// SIMATIC S7-200 SMART project (STEP 7-Micro/WIN SMART), CPU SR40

SYMBOL_TABLE 系统符号
Clock_1s         SM0.5    // 针对 1 s 的周期时间，时钟脉冲接通 0.5 s，断开 0.5 s.
END_SYMBOL_TABLE

ORGANIZATION_BLOCK MAIN:OB1
TITLE=程序注释
BEGIN
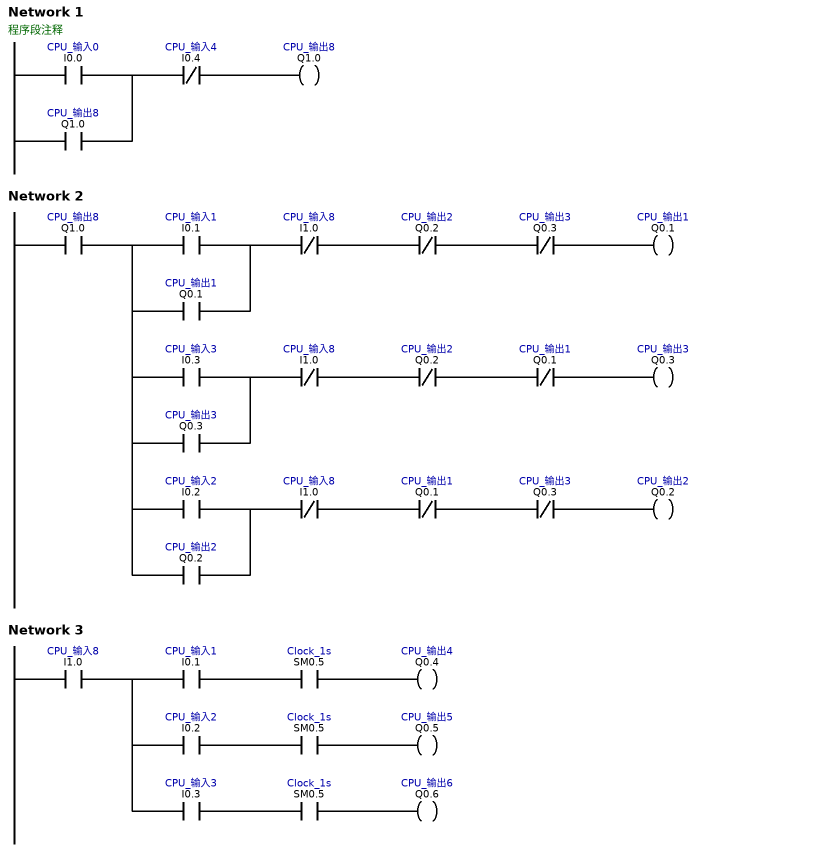
Network 1
// 程序段注释
LD     CPU_输入0:I0.0
O      CPU_输出8:Q1.0
AN     CPU_输入4:I0.4
=      CPU_输出8:Q1.0
Network 2
LD     CPU_输出8:Q1.0
LPS
LD     CPU_输入1:I0.1
O      CPU_输出1:Q0.1
ALD
AN     CPU_输入8:I1.0
AN     CPU_输出2:Q0.2
AN     CPU_输出3:Q0.3
=      CPU_输出1:Q0.1
LRD
LD     CPU_输入3:I0.3
O      CPU_输出3:Q0.3
ALD
AN     CPU_输入8:I1.0
AN     CPU_输出2:Q0.2
AN     CPU_输出1:Q0.1
=      CPU_输出3:Q0.3
LPP
LD     CPU_输入2:I0.2
O      CPU_输出2:Q0.2
ALD
AN     CPU_输入8:I1.0
AN     CPU_输出1:Q0.1
AN     CPU_输出3:Q0.3
=      CPU_输出2:Q0.2
Network 3
LD     CPU_输入8:I1.0
LPS
A      CPU_输入1:I0.1
A      Clock_1s:SM0.5
=      CPU_输出4:Q0.4
LRD
A      CPU_输入2:I0.2
A      Clock_1s:SM0.5
=      CPU_输出5:Q0.5
LPP
A      CPU_输入3:I0.3
A      Clock_1s:SM0.5
=      CPU_输出6:Q0.6
END_ORGANIZATION_BLOCK
